TYPE T_Type : __SYSTEM.TYPE_CLASS; END_TYPE

(* stored: Version 1.1.0.1
   DUT T_Type: Id {6586d12d-6f2c-0f59-00c5-531d107ef0be} *)
